(* PLC project SafeLOGIC-1, BrAutomation SafeDESIGNER  4.3.3.7 *)
(* stored: companyURL http://www.br-automation.com, creationDateTime Sat Nov 03 20:50:29 2018 *)

PROGRAM SP1130Sperre

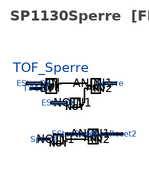
(* FBD diagram, written out as Structured Text *)
TOF_Sperre(IN := EStopOK, PT := T#12s);
Sperre := TOF_Sperre.Q AND NOT EStopOK;
EStopReset2 := EStopReset AND NOT Sperre;
END_PROGRAM
